// TIA Portal V21 export
DATA_BLOCK "ALARM"   // DB101
{ S7_Optimized_Access := 'FALSE' }
   VAR
      AL_EMG_STOP : Bool;
      AL_LOW_PRESSURE : Bool;
      AL_DOOR_OPEN : Bool;
      AL_DRUM_MTR_TRIP : Bool;
      AL_VACCUM_MTR_TRIP : Bool;
      AL_RECRC_TRIP : Bool;
      AL_PW_START : Bool;
      AL_PW_OVER : Bool;
      AL_WFI_START : Bool;
      AL_WFI_OVER : Bool;
      AL_STERILE_START : Bool;
      AL_STERILE_OVER : Bool;
      AL_DRY_START : Bool;
      AL_DRY_OVER : Bool;
      AL_PROCESS_COMP : Bool;
      AL_PRESSURE_HIGH : Bool;
      AL_RTD_FAIL : Bool;
      "AL_CHAMBER PRESS_FAIL" : Bool;
      "AL DOOR1 CLOSE LMT FAIL" : Bool;
      "AL DOOR2 CLOSE LMT FAIL" : Bool;
      "AL CHAMBER PRESS HIGH" : Bool;
      "AL JACKET RTD FAIL" : Bool;
      "AL BOILER TEMP HIGH" : Bool;
      "AL DOOR1 VCC FAIL" : Bool;
      "AL DOOR2 VCC FAIL" : Bool;
      "AL PHASE FAILURE" : Bool;
      "AL TEMP OVERSHOOT" : Bool;
      "AL CHAMBER RTD1 FAIL" : Bool;
      "AL CHAMBER RTD2 FAIL" : Bool;
      "AL CHAMBER RTD3 FAIL" : Bool;
      "AL CHAMBER RTD4 FAIL" : Bool;
      "AL JACKET PRESS FAIL" : Bool;
      "AL DOOR1 PRESS FAIL" : Bool;
      "AL DOOR2 PRESS FAIL" : Bool;
   END_VAR
BEGIN
END_DATA_BLOCK
